TYPE Task_1 :
	(
		NieuweOrderGaragist,
		VoorraadAdministratief,
		VerzamelingArtikelen,
		OrderGeanuleerd
	) := NieuweOrderGaragist;
END_TYPE

(* stored: Version 1.1.0.1, ProductVersion 3.1.4024.12
   DUT Task_1: Id {1b4acdbb-dead-4f52-ba94-f5c5c1cf4e46} *)
